PROGRAM OP60_Initialization_Seq
VAR
END_VAR

IF (SR60_Vert_servo_ctrl.Axis_In_Home)THEN
    OP60_Temp_hmeOK:=TRUE;
	OP60_HomeRunning:=FALSE;
	OP60_Homing_Seq:=0;
ELSE
	OP60_Temp_hmeOK:=FALSE;	
END_IF

CASE OP60_Homing_Seq OF
	0: IF (OP60_AutoSelected AND NOT OP60_HomeRunning AND NOT OP60_ErrorActive AND NOT  OP60_AutoRunning AND NOT OP60_StepRunning AND NOT OP60_Temp_hmeOK ) THEN
		OP60_HomeRunning:=TRUE;
		OP60_Homing_Seq:=10;	
	   END_IF
	10:IF (OP60_HomeRunning AND (OP60_HMI_Homing OR HMI_Reset))THEN 
		IF (SR60_Vert_servo_ctrl.Axis_In_Home) THEN 
			OP60_Homing_Seq:=20;
			SR60_Vert_servo_ctrl.Axis_Home_Cmd:=FALSE;
		ELSE
			SR60_Vert_servo_ctrl.Position:=0;
			SR60_Vert_servo_ctrl.Velocity:=100;			
			SR60_Vert_servo_ctrl.ABSmove_Start:=TRUE;
			SR60_Vert_servo_ctrl.Axis_Home_Cmd:=TRUE;
	    END_IF
	   END_IF		
	20:	OP60_Homing_Seq:=0;
		OP60_HomeRunning:=FALSE;
	
END_CASE

END_PROGRAM

(* stored: Version 1.1.0.1, ProductVersion 3.1.4024.11
   POU OP60_Initialization_Seq: Id {287c3516-f69b-446f-b67b-1719f3dc98a8}, SpecialFunc None *)
